FUNCTION_BLOCK A2X_AUI_MUX_3_UNGATED (* Wie A2X_AUI_MUX_3, aber OHNE Aenderungserkennung - reicht JEDES neu berechnete Ergebnis bedingungslos weiter (fuer Verbraucher, die eine periodische Kadenz unabhaengig von Wertaenderung brauchen, z.B. Ableitungs-/Frequenzberechnungen). (A2X multiplexor (generic FB)) *)
  (* Standard: 61499-2; Description: Copyright (c) 2026 Meisterschulen am Ostbahnhof This program and the accompanying materials are made available under the terms of the Eclipse Public License 2.0 which is available at https://www.eclipse.org/legal/epl-2.0/ SPDX-License-Identifier: EPL-2.0 *)
  (* Version 1.0, 2026-09-11, Franz Höpfinger, Meisterschulen am Ostbahnhof, A2X-Variante von AX_AUI_MUX_3_UNGATED - Adapter-Backend GEN_A2X_AUI_MUX noch zu implementieren. *)
  PACKAGE adapter::selection::unidirectional;
  {SET_ATTRIBUTE(eclipse4diac::core::GenericClassName, 'GEN_A2X_AUI_MUX')}
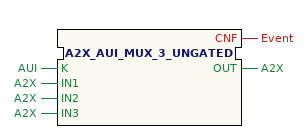
  EVENT_OUTPUT
    CNF; (* Confirmation of Set Index K *)
  END_EVENT
  SOCKETS
    K : adapter::types::unidirectional::AUI; (* index *)
    IN1 : adapter::types::unidirectional::A2X; (* Input value 1 (selected when K = 0) *)
    IN2 : adapter::types::unidirectional::A2X; (* Input value 2 (selected when K = 1) *)
    IN3 : adapter::types::unidirectional::A2X; (* Input value 3 (selected when K = 2) *)
  END_SOCKETS
  PLUGS
    OUT : adapter::types::unidirectional::A2X; (* IN1 for K = 0, IN2 for K = 1, IN3 for K = 2 *)
  END_PLUGS
END_FUNCTION_BLOCK
